// A discretized PID element. Transfer function:
// G(s) = Kp*(1+ (1/(Tn)) + (Tv/(1+Td)) )
FUNCTION_BLOCK FB_BasicPid EXTENDS ZigaLibs_Core.FB_HasTaskInfo
VAR_INPUT
	enable			: BOOL;		// Enables PID
	setpoint		: LREAL;	// Setpoint for PID controller when in ACTIVE moed
	manualSetpoint	: LREAL;	// Setpoint passed to output when MANUAL mode is active
	feedback		: LREAL;	// Feedback value for PID
	reset			: BOOL;		// Resets the controller
END_VAR
VAR_OUTPUT
	output	: LREAL;	// Output for the control variable, spanning from 0-100 (%) betwee Parameters.Minimum
	error	: BOOL;		// TRUE if error (incorrect parameters)
	errorId	: E_BasicPidErrorId;
END_VAR
VAR
	_parameters					: ST_PID_Parameters;
	_basicPid					: Tc2_Utilities.FB_BasicPID;
	_mode						: E_ControllerMode := E_ControllerMode.ACTIVE;
	_taskTimeAsSeconds			: LREAL;
	_modeChanged				: BOOL;
	_waitForControllerInRange	: BOOL;
	_setpointFromManualMode		: LREAL;
	_percentValueCurrent		: LREAL;
	_output						: LREAL;
END_VAR

error := FALSE;
IF THIS^.TaskInfo.CycleTime <> 0 THEN
	_taskTimeAsSeconds := 1000.0/DINT_TO_LREAL(THIS^.TaskInfo.CycleTime);	
END_IF


_basicPid.fKp := _parameters.Kp;
_basicPid.fTn := _parameters.Tn;
_basicPid.fTd := _parameters.Td;
_basicPid.fTv := _parameters.Tv;

IF _basicPid.fCtrlCycleTime = 0 OR (_parameters.CycleTime < _taskTimeAsSeconds) THEN
	IF _taskTimeAsSeconds <> 0 THEN
		// Set control time to a minimum of task cycle time
		_basicPid.fCtrlCycleTime := _taskTimeAsSeconds;
	ELSE
		// Cycle time invalid and can't be determined - exit
		errorId := E_BasicPidErrorId.INVALID_CYCLE_TIME;
		error := TRUE;
		output := 0;
		RETURN;
	END_IF
END_IF


IF NOT enable THEN
	_basicPid(
		bReset := NOT _basicPid.bReset, 
		fSetpointValue := 0, 
		fActualValue := 0);
	_output := 0;
	_waitForControllerInRange := FALSE;
ELSE
	CASE _mode OF
		E_ControllerMode.MANUAL:
			_output := MIN(_parameters.MaxOutput, MAX(0, manualSetpoint));
			_setpointFromManualMode := _output;
			_basicPid(
				bReset := NOT _basicPid.bReset, 
				fSetpointValue := 0, 
				fActualValue := 0);
		
		E_ControllerMode.ACTIVE:
			IF _modeChanged THEN
				_waitForControllerInRange := manualSetpoint <> 0;
			END_IF
			
			_basicPid(
				fActualValue := feedback,
				fSetpointValue := setpoint,
				bReset := FALSE);
				
			_percentValueCurrent := THIS^.ValueToPercentage(_basicPid.fCtrlOutput);
			
			// Wait for controller to reach the manual setpoint before activating it
			IF _waitForControllerInRange AND _parameters.ManualSwitchInRange <> 0.0 THEN
				IF (_percentValueCurrent + _parameters.ManualSwitchInRange) >= _setpointFromManualMode  THEN
					// Controller has reached the manual setpoint. Reset flag and instantly pass the value to output.
					_waitForControllerInRange := FALSE;
					_output := THIS^.ValueToPercentage(_basicPid.fCtrlOutput);
				ELSE
					// Wait for controller to reach the manual setpoint. Pass the last manual value until then.
					_output := _setpointFromManualMode;
				END_IF
			ELSE
				// Controller has reached the setpoint or the threshold is 0 - output is controlled by the PID
				_output := THIS^.ValueToPercentage(_basicPid.fCtrlOutput);
			END_IF
	END_CASE
END_IF

error := error OR _basicPid.nErrorStatus <> E_BasicPidErrorId.NO_ERROR;

CASE _basicPid.nErrorStatus OF
	0:
		errorId := E_BasicPidErrorId.NO_ERROR;
	1:
		errorId := E_BasicPidErrorId.INVALID_PARAMETERS;
	2:
		errorId := E_BasicPidErrorId.INVALID_CYCLE_TIME;
	ELSE
		errorId := E_BasicPidErrorId.UNKNOWN_ERROR;
END_CASE

output := _output;
_modeChanged := FALSE;

PROPERTY Mode : E_ControllerMode
GET
Mode := _mode;
END_GET
SET
IF _mode <> Mode THEN
	_modeChanged := TRUE;
END_IF

_mode := Mode;
END_SET
END_PROPERTY

{attribute 'monitoring' := 'variable'}
PROPERTY Parameters : REFERENCE TO ST_PID_Parameters
GET
Parameters REF= _parameters;
END_GET
SET
_parameters := Parameters;
END_SET
END_PROPERTY

// Calculates the percentage. Negative values are ommited and 0 is returned. Output is limited to _parameters.MaxOutput.
METHOD PRIVATE ValueToPercentage : LREAL
VAR_INPUT
	value	: LREAL;
END_VAR

VAR
	rangeSpan	: LREAL;
END_VAR
rangeSpan := (_parameters.ControllerUpperLimit - _parameters.ControllerLowerLimit);
IF value <= _parameters.ControllerLowerLimit OR rangeSpan <= 0THEN
	ValueToPercentage := 0.0;
	RETURN;
END_IF

ValueToPercentage := MIN((100.0 * (value / rangeSpan)), _parameters.MaxOutput);
END_METHOD

END_FUNCTION_BLOCK

(* stored: Version 1.1.0.1, ProductVersion 3.1.4024.16
   POU FB_BasicPid: Id {87a6a646-2e3c-0f51-25fc-4ebf8547d0b6}, SpecialFunc None
   Property Mode: Id {24964d76-0a70-017a-24fb-9b10e8cb23f7}
   Get Get: Id {1ae06da7-e4ee-039c-3b46-a4a35e441a56}
   Set Set: Id {f60bc4e9-596f-034f-26f5-28519fee7ec3}
   Property Parameters: Id {0caa46e7-f001-0916-0661-46965b0779f7}
   Get Get: Id {3d8d41e2-5643-09d5-26a1-5f61fc10e8b2}
   Set Set: Id {db7b6114-738d-0461-2d46-9e3a564bc534}
   Method ValueToPercentage: Id {b5bfe616-6fa1-04ce-071b-5d542c68b494} *)
